Staubli VAL3: ReplyCode.dtx

public num INVALID
public num SUCCESS
public num FAILURE
